# EPICS substitutions: tgpApp/Db/tpg26x.substitutions
file "tpgx6x.template" {
  pattern
    {P,    DEVICE, "IFPRESSUR1", "IFPRESSUR2", "PORT", "RECSIM", "DISABLE"}

    {"\$(P)", "TPG26x", "\$(IFPRESSUR1)", "\$(IFPRESSUR2)", "\$(PORT)", "\$(RECSIM)", "\$(DISABLE)"}
}
